TYPE "UDT_Fault_Word_0_System"
VERSION : 0.1
   STRUCT
      Safety_Relay_Refused : Bool;
      Safety_Relay_Tripped : Bool;
      Air_Pressure_Low : Bool;
      Src_Coolant_Flow_Low : Bool;
      Mag_Coolant_Flow_Low : Bool;
      Spare_0_5 : Bool;
      Spare_0_6 : Bool;
      Spare_0_7 : Bool;
      GateValve_Timeout : Bool;
      GateValve_Conflict : Bool;
      Spare_1_2 : Bool;
      Spare_1_3 : Bool;
      Spare_1_4 : Bool;
      Spare_1_5 : Bool;
      Spare_1_6 : Bool;
      Spare_1_7 : Bool;
      PC_Watchdog_Timeout : Bool;
      Remote_IO_Lost : Bool;
      Spare_2_2 : Bool;
      Spare_2_3 : Bool;
      Spare_2_4 : Bool;
      Spare_2_5 : Bool;
      Spare_2_6 : Bool;
      Spare_2_7 : Bool;
      Spare_3_0 : Bool;
      Spare_3_1 : Bool;
      Spare_3_2 : Bool;
      Spare_3_3 : Bool;
      Spare_3_4 : Bool;
      Spare_3_5 : Bool;
      Spare_3_6 : Bool;
      Spare_3_7 : Bool;
   END_STRUCT;
END_TYPE

TYPE "UDT_Fault_Word_1_Pumps"
VERSION : 0.1
   STRUCT
      Src_Turbo_Trip : Bool;
      Src_Turbo_Comms_Fail : Bool;
      Src_Turbo_Error_Active : Bool;
      Src_Turbo_Warning_Active : Bool;
      Spare_0_4 : Bool;
      Spare_0_5 : Bool;
      Spare_0_6 : Bool;
      Spare_0_7 : Bool;
      Ldlk_Turbo_Trip : Bool;
      Ldlk_Turbo_Comms_Fail : Bool;
      Ldlk_Turbo_Error_Active : Bool;
      Ldlk_Turbo_Warning_Active : Bool;
      Spare_1_4 : Bool;
      Spare_1_5 : Bool;
      Spare_1_6 : Bool;
      Spare_1_7 : Bool;
      Spare_2_0 : Bool;
      Spare_2_1 : Bool;
      Spare_2_2 : Bool;
      Spare_2_3 : Bool;
      Spare_2_4 : Bool;
      Spare_2_5 : Bool;
      Spare_2_6 : Bool;
      Spare_2_7 : Bool;
      Spare_3_0 : Bool;
      Spare_3_1 : Bool;
      Spare_3_2 : Bool;
      Spare_3_3 : Bool;
      Spare_3_4 : Bool;
      Spare_3_5 : Bool;
      Spare_3_6 : Bool;
      Spare_3_7 : Bool;
   END_STRUCT;
END_TYPE

TYPE "UDT_Fault_Word_2_Source"
VERSION : 0.1
   STRUCT
      Src_Body_Temp_High : Bool;
      Cesium_Oven_OverTemp : Bool;
      Cesium_Oven_HeatFail : Bool;
      Cesium_Oven_CoolFail : Bool;
      Filament_OverCurrent : Bool;
      Filament_OverVoltage : Bool;
      Filament_Fail : Bool;
      Spare_0_7 : Bool;
      Extraction_OverCurrent : Bool;
      Extraction_OverVoltage : Bool;
      Extraction_Fail : Bool;
      Extraction_Sustained_Arc : Bool;
      Spare_1_4 : Bool;
      Spare_1_5 : Bool;
      Spare_1_6 : Bool;
      Spare_1_7 : Bool;
      Target_OverCurrent : Bool;
      Target_OverVoltage : Bool;
      Target_Fail : Bool;
      Target_Sustained_Arc : Bool;
      Spare_2_4 : Bool;
      Spare_2_5 : Bool;
      Spare_2_6 : Bool;
      Spare_2_7 : Bool;
      Thermionic_OverCurrent : Bool;
      Thermionic_OverVoltage : Bool;
      Thermionic_Fail : Bool;
      Thermionic_Sustained_Arc : Bool;
      Spare_3_4 : Bool;
      Spare_3_5 : Bool;
      Spare_3_6 : Bool;
      Spare_3_7 : Bool;
   END_STRUCT;
END_TYPE

TYPE "UDT_Fault_Word_3_Spellman"
VERSION : 0.1
   STRUCT
      Unit1_Comms_Fail : Bool;
      Unit1_OverCurrent : Bool;
      Unit1_OverVoltage : Bool;
      Unit1_Fail : Bool;
      Unit1_Arc_Exceeded : Bool;
      Unit2_Comms_Fail : Bool;
      Unit2_OverCurrent : Bool;
      Unit2_OverVoltage : Bool;
      Unit2_Fail : Bool;
      Unit2_Arc_Exceeded : Bool;
      Unit3_Comms_Fail : Bool;
      Unit3_OverCurrent : Bool;
      Unit3_OverVoltage : Bool;
      Unit3_Fail : Bool;
      Unit3_Arc_Exceeded : Bool;
      Unit4_Comms_Fail : Bool;
      Unit4_OverCurrent : Bool;
      Unit4_OverVoltage : Bool;
      Unit4_Fail : Bool;
      Unit4_Arc_Exceeded : Bool;
      Unit5_Comms_Fail : Bool;
      Unit5_OverCurrent : Bool;
      Unit5_OverVoltage : Bool;
      Unit5_Fail : Bool;
      Unit5_Arc_Exceeded : Bool;
      Spare_3_1 : Bool;
      Spare_3_2 : Bool;
      Spare_3_3 : Bool;
      Spare_3_4 : Bool;
      Spare_3_5 : Bool;
      Spare_3_6 : Bool;
      Spare_3_7 : Bool;
   END_STRUCT;
END_TYPE

TYPE "UDT_Fault_Word_4_Magnet"
VERSION : 0.1
   STRUCT
      Magnet_Comms_Fail : Bool;
      Magnet_Short_Circuit : Bool;
      Magnet_Open_Circuit : Bool;
      Magnet_Unexpected_Res : Bool;
      Magnet_PSU_Overtemp : Bool;
      Magnet_PSU_PowerFail : Bool;
      Magnet_PSU_OVP : Bool;
      Magnet_PSU_OCP : Bool;
      Spare_1_0 : Bool;
      Spare_1_1 : Bool;
      Spare_1_2 : Bool;
      Spare_1_3 : Bool;
      Spare_1_4 : Bool;
      Spare_1_5 : Bool;
      Spare_1_6 : Bool;
      Spare_1_7 : Bool;
      Spare_2_0 : Bool;
      Spare_2_1 : Bool;
      Spare_2_2 : Bool;
      Spare_2_3 : Bool;
      Spare_2_4 : Bool;
      Spare_2_5 : Bool;
      Spare_2_6 : Bool;
      Spare_2_7 : Bool;
      Spare_3_0 : Bool;
      Spare_3_1 : Bool;
      Spare_3_2 : Bool;
      Spare_3_3 : Bool;
      Spare_3_4 : Bool;
      Spare_3_5 : Bool;
      Spare_3_6 : Bool;
      Spare_3_7 : Bool;
   END_STRUCT;
END_TYPE

TYPE "UDT_Fault_Word_5_Gauges"
VERSION : 0.1
   STRUCT
      Graphix_1_Comms_Fail : Bool;
      Graphix_2_Comms_Fail : Bool;
      VG1_Not_Found : Bool;
      VG1_Type_Mismatch : Bool;
      VG1_Above_SP_Warn : Bool;
      VG1_Rapid_Rise_Warn : Bool;
      VG2_Not_Found : Bool;
      VG2_Type_Mismatch : Bool;
      VG2_Above_SP_Warn : Bool;
      VG2_Rapid_Rise_Warn : Bool;
      VG3_Not_Found : Bool;
      VG3_Type_Mismatch : Bool;
      VG3_Above_SP_Warn : Bool;
      VG3_Rapid_Rise_Warn : Bool;
      VG4_Not_Found : Bool;
      VG4_Type_Mismatch : Bool;
      VG4_Above_SP_Warn : Bool;
      VG4_Rapid_Rise_Warn : Bool;
      VG5_Not_Found : Bool;
      VG5_Type_Mismatch : Bool;
      VG5_Above_SP_Warn : Bool;
      VG5_Rapid_Rise_Warn : Bool;
      VG6_Not_Found : Bool;
      VG6_Type_Mismatch : Bool;
      VG6_Above_SP_Warn : Bool;
      VG6_Rapid_Rise_Warn : Bool;
      Spare_3_2 : Bool;
      Spare_3_3 : Bool;
      Spare_3_4 : Bool;
      Spare_3_5 : Bool;
      Spare_3_6 : Bool;
      Spare_3_7 : Bool;
   END_STRUCT;
END_TYPE

